{attribute addProperty BoxType "AT2050-0500-0022"}
{attribute addProperty Id "A_0091_AT2020_5250_0017_AT2020_5250AT2020_3DCFC8D064080"}
{attribute addProperty CRC "502046396"}
{attribute addProperty SizeInBites "640"}
{attribute addProperty SizeInBytes "80"}
TYPE A_0053_AT2050_0500_0022_1DEC9EBC EXTENDS AT2050_9506A482 :
STRUCT
	{attribute addProperty Name "A_0091_AT2020_5250_0017_AT2020_5250"}
	A_0091_AT2020_5250_0017_AT2020_5250 : AT2020_3DCFC8D0;
END_STRUCT
END_TYPE

(* stored: Version 1.2.0.0, ProductVersion 3.1.4024.9
   DUT A_0053_AT2050_0500_0022_1DEC9EBC: Id {440f8891-88fc-47a9-bae9-8d16210f10c9} *)
